Fanuc KAREL source: kt00329.KL

-- PROVISIONAL review KL for V770-1; original PC SHA256 aac8426b47d65597a73d19eb2bfcd480f0b6f45c644cd19e516790f00347c8da
-- Incomplete behavior may be omitted. Consult companion uncertainty JSON. Do not deploy.
PROGRAM KT00329
%NOLOCKGROUP
VAR
  I1 : INTEGER
  I2 : INTEGER
  OUT : BOOLEAN
BEGIN
  -- UNRESOLVED_PC offsets 5-16; opcodes 2E,23
  -- UNRESOLVED_PC offsets 21-32; opcodes 2E,23
  -- UNRESOLVED_PC offsets 37-48; opcodes 2E,23
  -- UNRESOLVED_PC offsets 53-64; opcodes 2E,23
  -- UNRESOLVED_PC offsets 69-88; opcodes 21,21,59,23
  -- UNRESOLVED_PC offsets 93-97; opcodes 7F
END KT00329
